FUNCTION GetAnyType : __SYSTEM.AnyType
VAR_INPUT
	object		: ANY;
END_VAR

GetAnyType := object;

END_FUNCTION

(* stored: Version 1.1.0.1
   POU GetAnyType: Id {174e1356-f49a-01e1-2125-3395432c8939}, SpecialFunc None *)
